// TIA Portal V19 export
TYPE "dtTimerArguments"
   STRUCT
      sec { S7_SetPoint := 'True'} : USInt;   // seconds
      min { S7_SetPoint := 'True'} : USInt;   // minutes
      hour { S7_SetPoint := 'True'} : UInt;   // hours
   END_STRUCT;
END_TYPE
